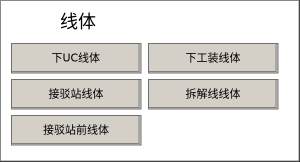
VISUALIZATION CtrlLine  // 300x162
    RoundedRectangle (0,0 300x162)
    Label (13,7 130x30), "线体"
    Button (11,43 130x30), "下UC线体"
        toggle GVL.arrFbLine[E_LineAxis.UnloadUc].Execute.bManual
    Button (148,43 130x30), "下工装线体"
        toggle GVL.arrFbLine[E_LineAxis.UnloadForck].Execute.bManual
    Button (11,79 130x30), "接驳站线体"
        toggle GVL.arrFbLine[E_LineAxis.Acquire].Execute.bManual
    Button (148,79 130x30), "拆解线线体"
        toggle GVL.arrFbLine[E_LineAxis.Dismantling].Execute.bManual
    Button (11,115 130x30), "接驳站前线体"
        toggle GVL.arrFbLine[E_LineAxis.AcquireFront].Execute.bManual
END_VISUALIZATION

(* stored: Version 1.1.0.1, ProductVersion 3.1.4024.3
   Visu CtrlLine: Id {fe176b47-f187-4c6a-9336-8e4c0993602f} *)
